// Mitsubishi GX Works2 project: 20141114音声   PLC: FX1N/FX1NC

PROGRAM MAIN
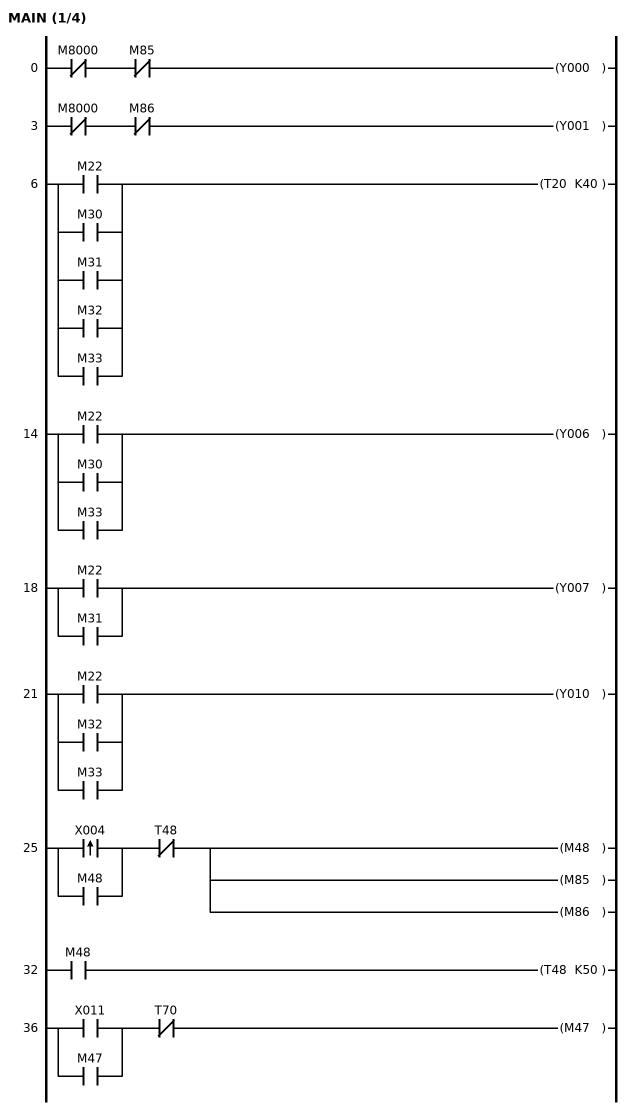
0     LDI     M8000
      ANI     M85
      OUT     Y000
3     LDI     M8000
      ANI     M86
      OUT     Y001
6     LD      M22
      OR      M30
      OR      M31
      OR      M32
      OR      M33
      OUT     T20 K40
14    LD      M22
      OR      M30
      OR      M33
      OUT     Y006
18    LD      M22
      OR      M31
      OUT     Y007
21    LD      M22
      OR      M32
      OR      M33
      OUT     Y010
25    LDP     X004
      OR      M48
      ANI     T48
      OUT     M48
      OUT     M85
      OUT     M86
32    LD      M48
      OUT     T48 K50
36    LD      X011
      OR      M47
      ANI     T70
      OUT     M47
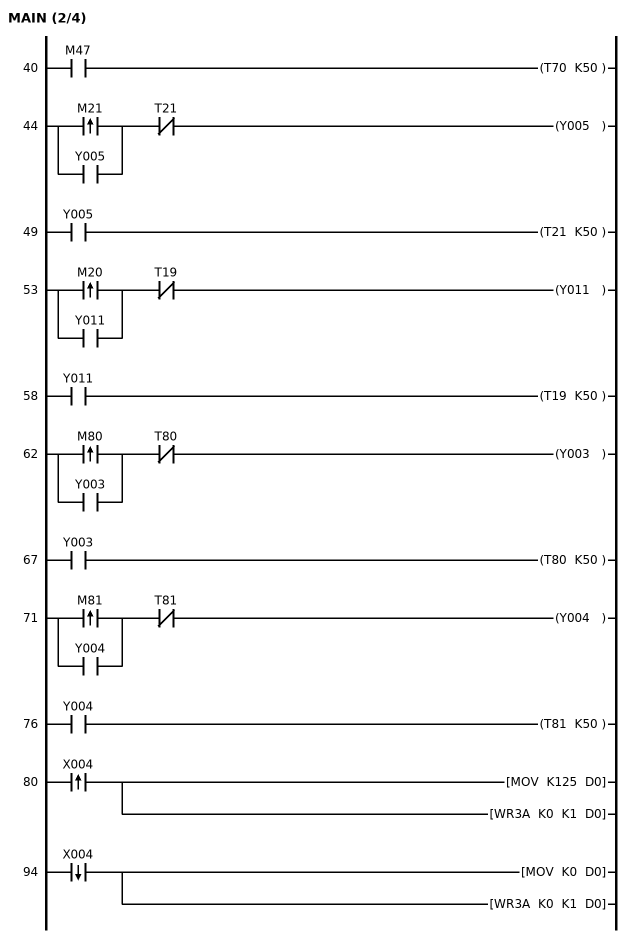
40    LD      M47
      OUT     T70 K50
44    LDP     M21
      OR      Y005
      ANI     T21
      OUT     Y005
49    LD      Y005
      OUT     T21 K50
53    LDP     M20
      OR      Y011
      ANI     T19
      OUT     Y011
58    LD      Y011
      OUT     T19 K50
62    LDP     M80
      OR      Y003
      ANI     T80
      OUT     Y003
67    LD      Y003
      OUT     T80 K50
71    LDP     M81
      OR      Y004
      ANI     T81
      OUT     Y004
76    LD      Y004
      OUT     T81 K50
80    LDP     X004
      MOV     K125 D0
      WR3A    K0 K1 D0
94    LDF     X004
      MOV     K0 D0
      WR3A    K0 K1 D0
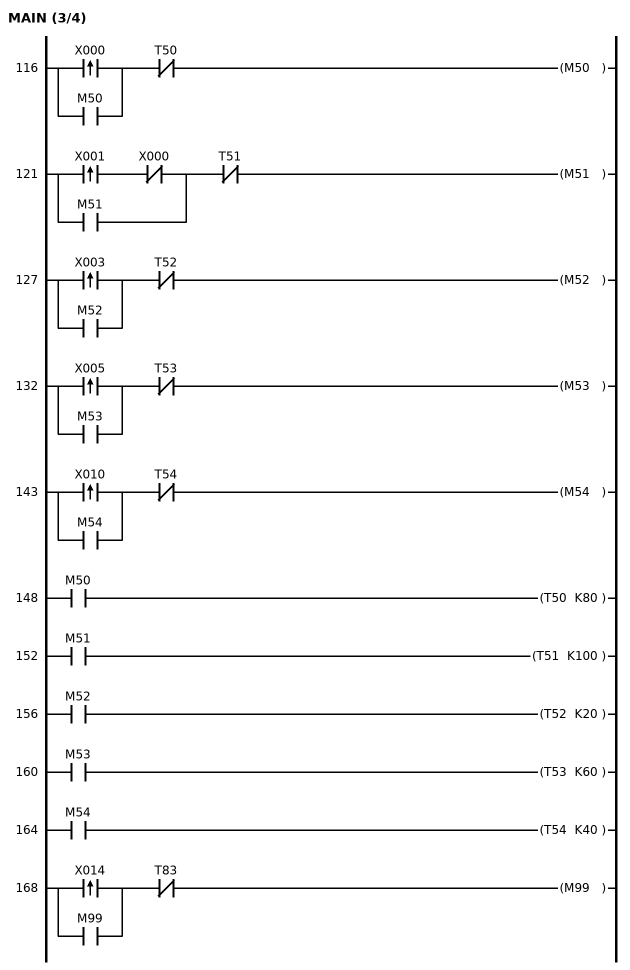
116   LDP     X000
      OR      M50
      ANI     T50
      OUT     M50
121   LDP     X001
      ANI     X000
      OR      M51
      ANI     T51
      OUT     M51
127   LDP     X003
      OR      M52
      ANI     T52
      OUT     M52
132   LDP     X005
      OR      M53
      ANI     T53
      OUT     M53
143   LDP     X010
      OR      M54
      ANI     T54
      OUT     M54
148   LD      M50
      OUT     T50 K80
152   LD      M51
      OUT     T51 K100
156   LD      M52
      OUT     T52 K20
160   LD      M53
      OUT     T53 K60
164   LD      M54
      OUT     T54 K40
168   LDP     X014
      OR      M99
      ANI     T83
      OUT     M99
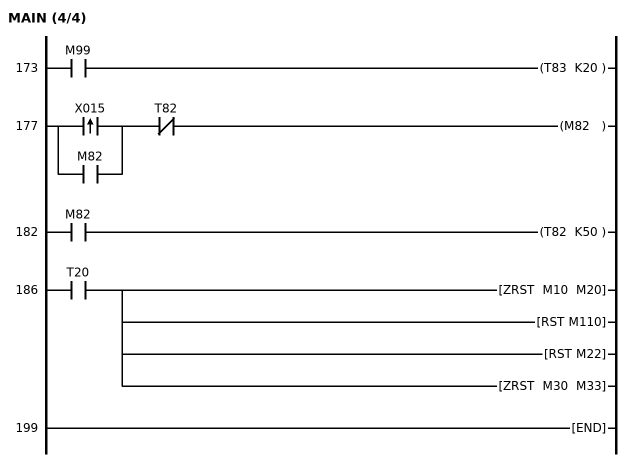
173   LD      M99
      OUT     T83 K20
177   LDP     X015
      OR      M82
      ANI     T82
      OUT     M82
182   LD      M82
      OUT     T82 K50
186   LD      T20
      ZRST    M10 M20
      RST     M110
      RST     M22
      ZRST    M30 M33
199   END
END_PROGRAM
